FUNCTION_BLOCK FB_Input IMPLEMENTS I_Input
VAR_INPUT
END_VAR
VAR_OUTPUT
END_VAR
VAR
	sDescription			:	STRING; //Description of the physical input
	bIn				AT %I*	:	BOOL;	// Physical input
	bRisingTrigger			:	BOOL;
	bFallingTrigger			:	BOOL;
	rtIn					:	R_TRIG; //Rising edge of the input
	ftIn					:	F_TRIG; //Falling edge of the input	
END_VAR

PROPERTY Description : STRING
GET
Description := sDescription;
END_GET
SET
sDescription := Description;
END_SET
END_PROPERTY

PROPERTY Value : BOOL
GET
Value := bIn;
END_GET
END_PROPERTY

END_FUNCTION_BLOCK

(* stored: Version 1.1.0.1, ProductVersion 3.1.4024.12
   POU FB_Input: Id {223e9000-979a-4a8f-8fcf-710a846d6047}, SpecialFunc None
   Property Description: Id {057ffb6c-b47d-4542-ada6-dd39a07962e6}
   Get Get: Id {664afd07-53a4-4737-b46e-9eee8e2442b4}
   Set Set: Id {35cb0eae-5527-43e8-b4fc-212a882f116c}
   Property Value: Id {a95c409d-bb64-41c3-acde-78b674b539d7}
   Get Get: Id {96c92c67-f86b-4d16-a169-fc13b9bd4a26} *)
